{attribute 'qualified_only'}
{attribute 'strict'}
TYPE E_DB_QUERY_STATE :
(
	IDLE_STATE,
	SELECT_POST_LAST_RUN,
	INSERT_RUN,
	SELECT_LAST_CALIBRATION_ID,
	INSERT_CALIBRATION_VALUES,
	INSERT_CALIBRATION,
	SELECT_LAST_SYSTEM_ID,
	SELECT_ALL_SYSTEM,
	INSERT_SYS_PARAMETERS,
	SELECT_ALL_METHODS,
	SELECT_ALL_ACTV_METHODS,
	SELECT_WHOLE_METHODS,
	INSERT_NEW_METHOD,
	UPDATE_DEACTV_METHOD,
	SELECT_LAST_METHOD_ID,
	SELECT_VOLUME_DATA,
	INSERT_VOLUME_DATA,
	SELECT_ALL_CURRENT_USERS,
	SELECT_ALL_USERS,
	SELECT_LAST_SOLVENT,
	SELECT_ALL_SOLVENT,
	INSERT_SOLVENT,
	INSERT_LINEAR_MOTORS,
	SELECT_LINEAR_MOTORS,
	SELECT_LAST_CALIBRATION,
	SELECT_CALIB_REPORT_LIST,
	SELECT_CALIB_REPORT_DETAILS,
	SELECT_SYSTEM_REPORT_LIST,
	SELECT_SYSTEM_REPORT_DETAILS,
	SELECT_POSTRUN_REPORT_LIST,
	SELECT_POSTRUN_REPORT_DETAILS,
	DELETE_CALIBRATION_HEAD,
	SELECT_CALIB_REPORT_BY_ID,
	SELECT_CALIB_REPORT_VALUES_BY_ID,
	SELECT_SYSTEM_SETTINGS_REPORT_LIST,
	SELECT_SYSTEM_SETTINGS_BY_ID,
	SELECT_METHOD_REPORT_SEARCH,
	SELECT_METHOD_REPORT_LIST,
	SELECT_RUN_REPORT_LIST,
	SELECT_RECIPE_HEADER_BY_ID,
	SELECT_RECIPE_VOLUME_BY_ID,
	SELECT_POSTRUN_RUN_BY_ID,
	SELECT_POSTRUN_METHOD_BY_RUN_ID,
	SELECT_POSTRUN_VOLUME_BY_METHOD_ID,
	SELECT_LINEAR_BY_ID,
	SELECT_LINEAR_REPORT_SEARCH,
	SELECT_LAST_LINEAR_REPORT,
	SELECT_LAST_POSTRUN_RUN,
	SELECT_LAST_PUMP_CALIBRATION,
	SELECT_SYSTEM_HISTORY_REPORT,
	SELECT_LINEAR_HISTORY_REPORT,
	SELECT_COMPLETE_METHOD_REPORT,
	SELECT_COMPLETE_METHOD_REPORT_VOLUMES,
	INSERT_USER,
	INSERT_USER_MGMT_HISTORY,
	ERROR_STATE
);
END_TYPE

(* stored: Version 1.1.0.1, ProductVersion 3.1.4024.15
   EnumerationTextList E_DB_QUERY_STATE: Id {e636e289-9b0b-435f-a6f8-55952d4015dd} *)
